# EPICS autosave request: ADApp/Db/mar345_settings.req
$(P)$(R)EraseMode
$(P)$(R)NumErase
$(P)$(R)ScanSize
$(P)$(R)ScanResolution
